INTERFACE I_ContinuousDrive

METHOD atHome : BOOL
VAR_INPUT
END_VAR
END_METHOD

METHOD hasError : BOOL
VAR_INPUT
END_VAR
END_METHOD

METHOD ABSTRACT homingSequence : BOOL
VAR_INPUT
END_VAR
END_METHOD

METHOD isBusy : BOOL
VAR_INPUT
END_VAR
END_METHOD

METHOD moveContinuous : BOOL
VAR_INPUT
	direction : MC_Direction;
END_VAR
END_METHOD

END_INTERFACE

(* stored: Version 1.1.0.1, ProductVersion 3.1.4024.11
   Itf I_ContinuousDrive: Id {27e7ee41-ea84-43ba-bbab-fcee94cc798c}
   Folder Get: Id {8e563fc4-6509-46e4-bd24-3ba5395a885c}
   Method atHome: Id {97ea62c5-7480-4d22-8b85-ba8010c5ba9e}
   Method hasError: Id {a9d197f0-48b9-4496-8069-a8fb6762a8d6}
   Method homingSequence: Id {26d9704b-2987-4774-98e0-6bd9116c3ba7}
   Method isBusy: Id {583782d4-4232-4857-83f8-f587195608f9}
   Method moveContinuous: Id {aab498f2-15fd-447c-8469-faaeaeb26562} *)
